(* Logix 5000 project; controller PLC_AutoSeats Emulate 5570 rev 30.12; software revision 30.00 *)

TASK MainTask (continuous, watchdog 500 ms) : MainProgram

MODULES
   Local : Emulate 5570 (ICP 2, rev 30.12)
END_MODULES

VAR_GLOBAL   (* controller tags *)
   Active_PP : BOOL;
   Active_PU : BOOL;
   Active_Soldadura : BOOL;
   Auto : BOOL;
   Emer_Stop_SCADA_PP : BOOL;
   Emer_Stop_SCADA_PU : BOOL;
   Emer_Stop_SCADA_Soldadura : BOOL;
   Estado_PP : DINT;
   Estado_PU : DINT;
   Estado_Soldadura : DINT;
   Mantenimiento_PP : BOOL;
   Mantenimiento_PU : BOOL;
   Mantenimiento_Soldadura : BOOL;
   Manual : BOOL := 1;
   Modo_Op : DINT;
   OSF_01 : BOOL;
   OSF_02 : BOOL;
   OSF_OB_01 : BOOL;
   OSF_OB_02 : BOOL;
   OSR_01 : BOOL;
   OSR_02 : BOOL;
   OSR_03 : BOOL;
   OSR_04 : BOOL;
   OSR_05 : BOOL;
   OSR_06 : BOOL;
   OSR_07 : BOOL;
   OSR_08 : BOOL;
   OSR_09 : BOOL;
   OSR_OB_01 : BOOL;
   OSR_OB_02 : BOOL;
   OSR_OB_03 : BOOL;
   OSR_OB_04 : BOOL;
   OSR_OB_05 : BOOL;
   OSR_OB_06 : BOOL;
   OSR_OB_07 : BOOL;
   OSR_OB_08 : BOOL;
   OSR_OB_09 : BOOL;
   Parar_Ciclo_PP : BOOL;
   Parar_Ciclo_PU : BOOL;
   Parar_Ciclo_Soldadura : BOOL;
   PP_Banda : BOOL;
   PP_Gen_Reposabrazo : BOOL;
   PP_Mover_Molde : BOOL;
   PP_Pos_Molde : REAL;
   PP_Resistencia : BOOL;
   PP_Sensor_Banda_Salida : BOOL;
   PP_Sensor_Molde_Abierto : BOOL;
   PP_Sensor_Molde_Cerrado : BOOL;
   PP_Step1 : BOOL;
   PP_Step2 : BOOL;
   PP_Step3 : BOOL;
   PP_Step4 : BOOL;
   PP_Step5 : BOOL;
   PP_Step6 : BOOL;
   PP_Step7 : BOOL;
   PP_Step8 : BOOL;
   PP_Tornillo_Ext : DINT;
   Producto : DINT;
   PU_Act_Eyector : BOOL;
   PU_Act_Inyector : BOOL;
   PU_Sensor_Pos_MC_1 : DINT;
   PU_Sensor_Pos_MC_2 : DINT;
   PU_Sensor_Pos_ME_1 : DINT;
   PU_Sensor_Pos_ME_2 : DINT;
   PU_Sensor_Pos_R1 : DINT;
   PU_Sensor_Pos_R2 : DINT;
   PU_Sensor_Pos_R3 : DINT;
   Soldadura_Banda_Entrada : BOOL;
   Soldadura_Banda_Salida : BOOL;
   Soldadura_Eli_Marco_Salida : BOOL;
   Soldadura_Eli_Material_Entrada : BOOL;
   Soldadura_Gen_Marco_Salida : BOOL;
   Soldadura_Gen_Material_Entrada : BOOL;
   Soldadura_Giro_0_Listo : BOOL;
   Soldadura_Giro_180_Listo : BOOL;
   Soldadura_Giro_Listo : BOOL;
   Soldadura_Matriz : DINT;
   Soldadura_Primera_Listo : BOOL;
   Soldadura_Segunda_Listo : BOOL;
   Soldadura_Sensor_Entrada : BOOL;
   Soldadura_Sensor_Entrada_Aux : BOOL;
   Soldadura_Sensor_Pos_Matriz : DINT;
   Soldadura_Sensor_Salida : BOOL;
   Soldadura_Sensor_Salida_Aux : BOOL;
   Soldadura_Start_Operario : BOOL;
   Soldadura_Step1 : BOOL;
   Soldadura_Step2 : BOOL;
   Soldadura_Step3 : BOOL;
   Soldadura_Step4 : BOOL;
   Soldadura_Step5 : BOOL;
   Soldadura_Step6 : BOOL;
   Soldadura_Step7 : BOOL;
   Soldadura_Step8 : BOOL;
   Soldadura_Step9 : BOOL;
   Start_Fisico_PP : BOOL;   // Boton Verde Fisico
   Start_Fisico_PU : BOOL;
   Start_Fisico_Soldadura : BOOL;
   Start_SCADA_PP : BOOL;
   Start_SCADA_PU : BOOL;
   Start_SCADA_Soldadura : BOOL;
   Start_Telegram_PP : BOOL;
   Start_Telegram_PU : BOOL;
   Start_Telegram_Soldadura : BOOL;
   Stop_Fisico_PP : BOOL;
   Stop_Fisico_PU : BOOL;
   Stop_Fisico_Soldadura : BOOL;
   Stop_SCADA_PP : BOOL;
   Stop_SCADA_PU : BOOL;
   Stop_SCADA_Soldadura : BOOL;
   Stop_Telegram_PU : BOOL;
   Temp_PP : BOOL;
   Temp_PU : BOOL;
   Temp_Soldadura : BOOL;
   TOF_01 : TIMER := (PRE := 1000);
   TOF_02 : TIMER := (PRE := 1000);
   TOF_03 : TIMER := (PRE := 1000);
   TOF_04 : TIMER := (PRE := 3000);
   TOF_05 : TIMER := (PRE := 1000);
   TOF_06 : TIMER := (PRE := 1000);
   TOF_07 : TIMER := (PRE := 3000);
   TOF_08 : TIMER := (PRE := 1000);
   TON_01 : TIMER := (PRE := 8000);
   TON_02 : TIMER := (PRE := 10000);
   TON_03 : TIMER := (PRE := 10000);
   TON_04 : TIMER := (PRE := 7500);
   TON_05 : TIMER := (PRE := 5000);
END_VAR

PROGRAM MainProgram   (* main routine MainRoutine *)

ROUTINE Celda_Inyeccion_PP   (* ladder *)
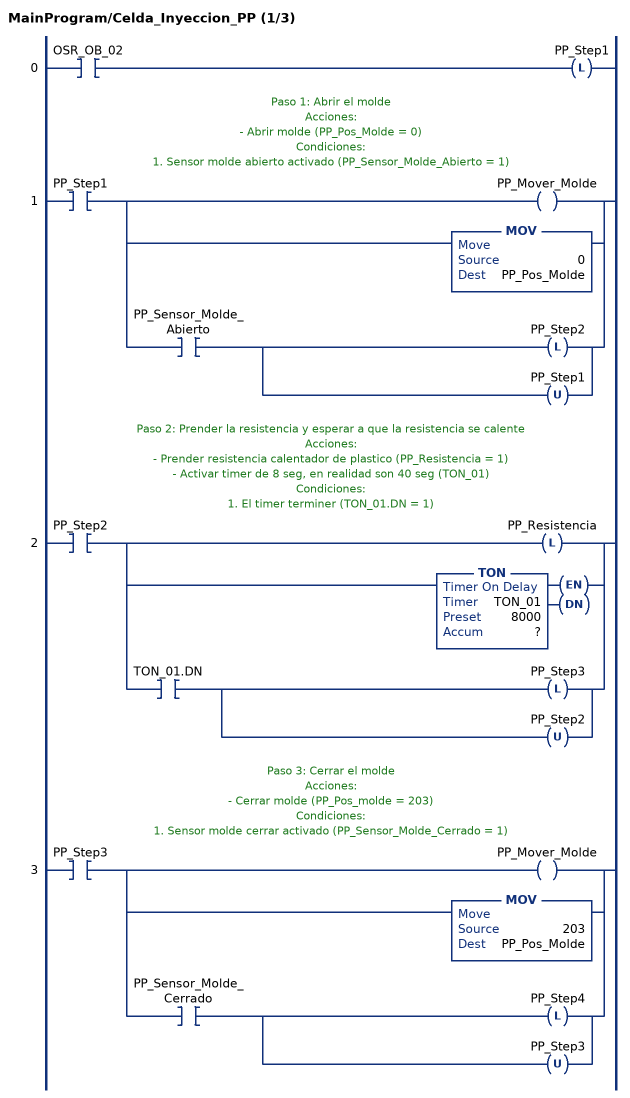
   0: XIC(OSR_OB_02)OTL(PP_Step1);
   // Paso 1: Abrir el molde
   // Acciones:
   // - Abrir molde (PP_Pos_Molde = 0)
   // Condiciones:
   // 1. Sensor molde abierto activado (PP_Sensor_Molde_Abierto = 1)
   1: XIC(PP_Step1)[[OTE(PP_Mover_Molde) ,MOV(0,PP_Pos_Molde) ] ,XIC(PP_Sensor_Molde_Abierto) [OTL(PP_Step2) ,OTU(PP_Step1) ] ];
   // Paso 2: Prender la resistencia y esperar a que la resistencia se calente
   // Acciones:
   // - Prender resistencia calentador de plastico (PP_Resistencia = 1)
   // - Activar timer de 8 seg, en realidad son 40 seg (TON_01)
   // Condiciones:
   // 1. El timer terminer (TON_01.DN = 1)
   2: XIC(PP_Step2)[[OTL(PP_Resistencia) ,TON(TON_01,?,?) ] ,XIC(TON_01.DN) [OTL(PP_Step3) ,OTU(PP_Step2) ] ];
   // Paso 3: Cerrar el molde
   // Acciones:
   // - Cerrar molde (PP_Pos_molde = 203)
   // Condiciones:
   // 1. Sensor molde cerrar activado (PP_Sensor_Molde_Cerrado = 1)
   3: XIC(PP_Step3)[[OTE(PP_Mover_Molde) ,MOV(203,PP_Pos_Molde) ] ,XIC(PP_Sensor_Molde_Cerrado) [OTL(PP_Step4) ,OTU(PP_Step3) ] ];
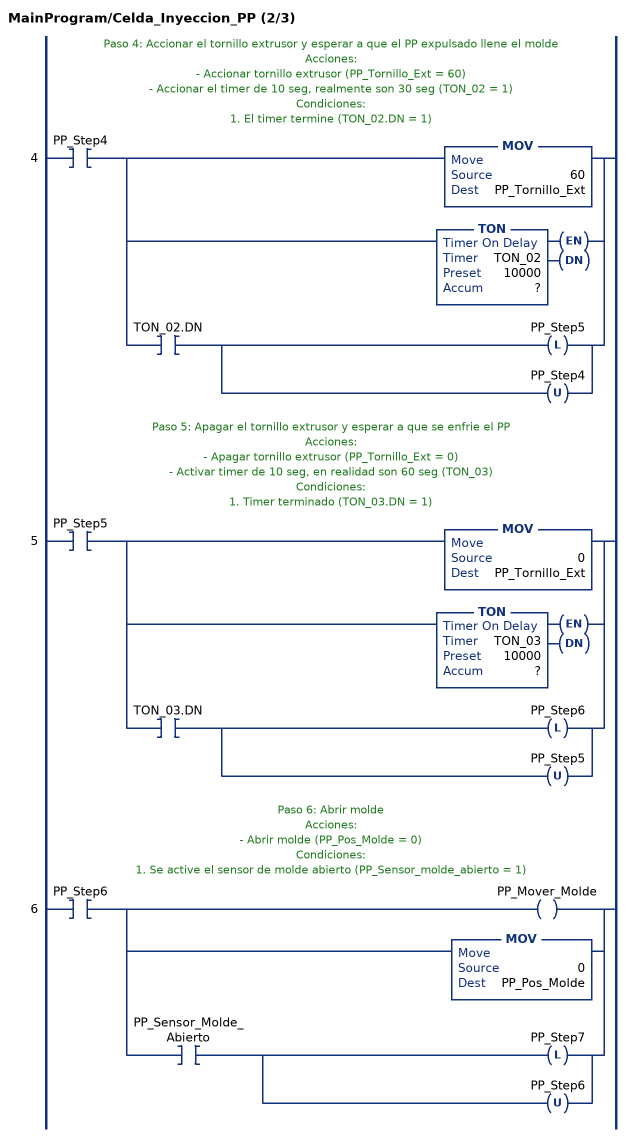
   // Paso 4: Accionar el tornillo extrusor y esperar a que el PP expulsado llene el molde
   // Acciones:
   // - Accionar tornillo extrusor (PP_Tornillo_Ext = 60)
   // - Accionar el timer de 10 seg, realmente son 30 seg (TON_02 = 1)
   // Condiciones:
   // 1. El timer termine (TON_02.DN = 1)
   4: XIC(PP_Step4)[[MOV(60,PP_Tornillo_Ext) ,TON(TON_02,?,?) ] ,XIC(TON_02.DN) [OTL(PP_Step5) ,OTU(PP_Step4) ] ];
   // Paso 5: Apagar el tornillo extrusor y esperar a que se enfrie el PP
   // Acciones:
   // - Apagar tornillo extrusor (PP_Tornillo_Ext = 0)
   // - Activar timer de 10 seg, en realidad son 60 seg (TON_03)
   // Condiciones:
   // 1. Timer terminado (TON_03.DN = 1)
   5: XIC(PP_Step5)[[MOV(0,PP_Tornillo_Ext) ,TON(TON_03,?,?) ] ,XIC(TON_03.DN) [OTL(PP_Step6) ,OTU(PP_Step5) ] ];
   // Paso 6: Abrir molde
   // Acciones:
   // - Abrir molde (PP_Pos_Molde = 0)
   // Condiciones:
   // 1. Se active el sensor de molde abierto (PP_Sensor_molde_abierto = 1)
   6: XIC(PP_Step6)[[OTE(PP_Mover_Molde) ,MOV(0,PP_Pos_Molde) ] ,XIC(PP_Sensor_Molde_Abierto) [OTL(PP_Step7) ,OTU(PP_Step6) ] ];
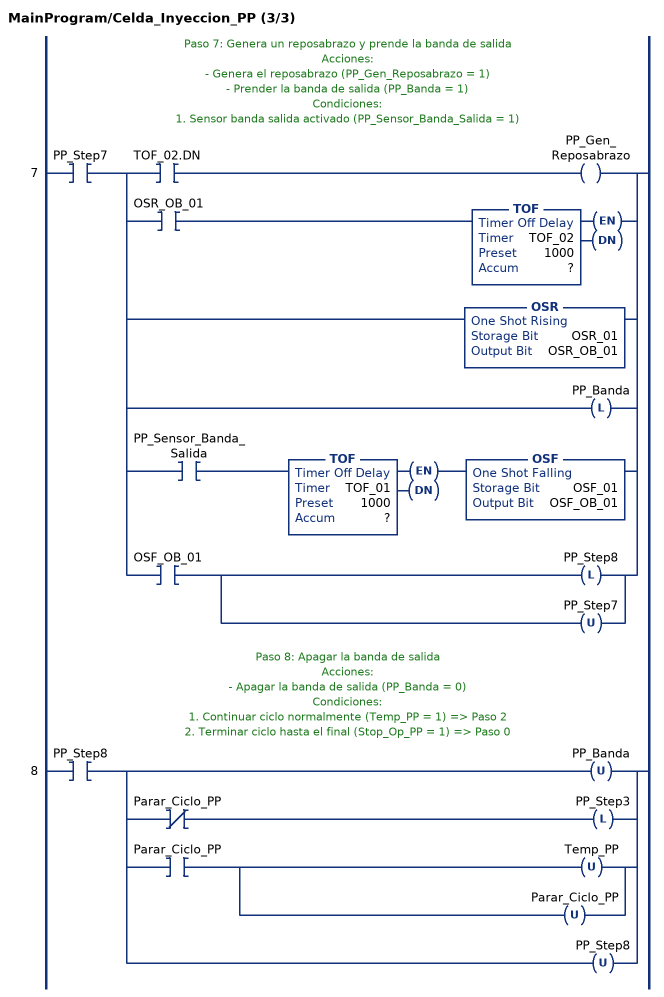
   // Paso 7: Genera un reposabrazo y prende la banda de salida
   // Acciones:
   // - Genera el reposabrazo (PP_Gen_Reposabrazo = 1)
   // - Prender la banda de salida (PP_Banda = 1)
   // Condiciones:
   // 1. Sensor banda salida activado (PP_Sensor_Banda_Salida = 1)
   7: XIC(PP_Step7)[[[[XIC(TOF_02.DN) OTE(PP_Gen_Reposabrazo) ,XIC(OSR_OB_01) TOF(TOF_02,?,?) ] ,OSR(OSR_01,OSR_OB_01) ] ,[OTL(PP_Banda) ,XIC(PP_Sensor_Banda_Salida) TOF(TOF_01,?,?) OSF(OSF_01,OSF_OB_01) ] ] ,XIC(OSF_OB_01) [OTL(PP_Step8) ,OTU(PP_Step7) ] ];
   // Paso 8: Apagar la banda de salida
   // Acciones:
   // - Apagar la banda de salida (PP_Banda = 0)
   // Condiciones:
   // 1. Continuar ciclo normalmente (Temp_PP = 1) => Paso 2
   // 2. Terminar ciclo hasta el final (Stop_Op_PP = 1) => Paso 0
   8: XIC(PP_Step8)[OTU(PP_Banda) ,[[XIO(Parar_Ciclo_PP) OTL(PP_Step3) ,XIC(Parar_Ciclo_PP) [OTU(Temp_PP) ,OTU(Parar_Ciclo_PP) ] ] ,OTU(PP_Step8) ] ];
END_ROUTINE

ROUTINE Celda_Soldadura   (* ladder *)
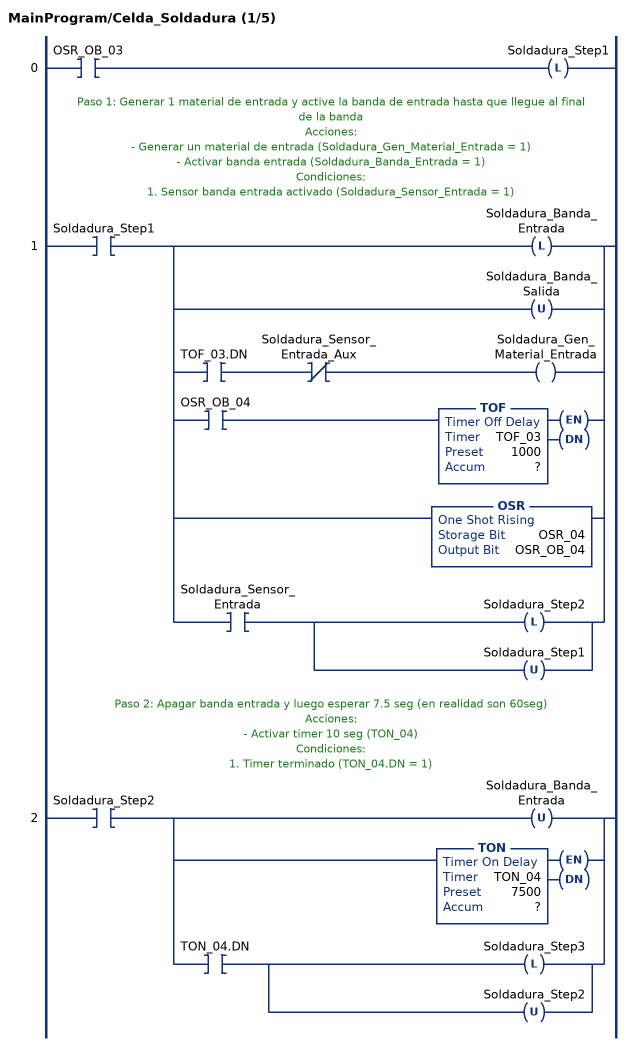
   0: XIC(OSR_OB_03)OTL(Soldadura_Step1);
   // Paso 1: Generar 1 material de entrada y active la banda de entrada hasta que llegue al final de la banda
   // Acciones:
   // - Generar un material de entrada (Soldadura_Gen_Material_Entrada = 1)
   // - Activar banda entrada (Soldadura_Banda_Entrada = 1)
   // Condiciones:
   // 1. Sensor banda entrada activado (Soldadura_Sensor_Entrada = 1)
   1: XIC(Soldadura_Step1)[[[OTL(Soldadura_Banda_Entrada) ,OTU(Soldadura_Banda_Salida) ] ,[XIC(TOF_03.DN) XIO(Soldadura_Sensor_Entrada_Aux) OTE(Soldadura_Gen_Material_Entrada) ,[XIC(OSR_OB_04) TOF(TOF_03,?,?) ,OSR(OSR_04,OSR_OB_04) ] ] ] ,XIC(Soldadura_Sensor_Entrada) [OTL(Soldadura_Step2) ,OTU(Soldadura_Step1) ] ];
   // Paso 2: Apagar banda entrada y luego esperar 7.5 seg (en realidad son 60seg)
   // Acciones:
   // - Activar timer 10 seg (TON_04)
   // Condiciones:
   // 1. Timer terminado (TON_04.DN = 1)
   2: XIC(Soldadura_Step2)[[OTU(Soldadura_Banda_Entrada) ,TON(TON_04,?,?) ] ,XIC(TON_04.DN) [OTL(Soldadura_Step3) ,OTU(Soldadura_Step2) ] ];
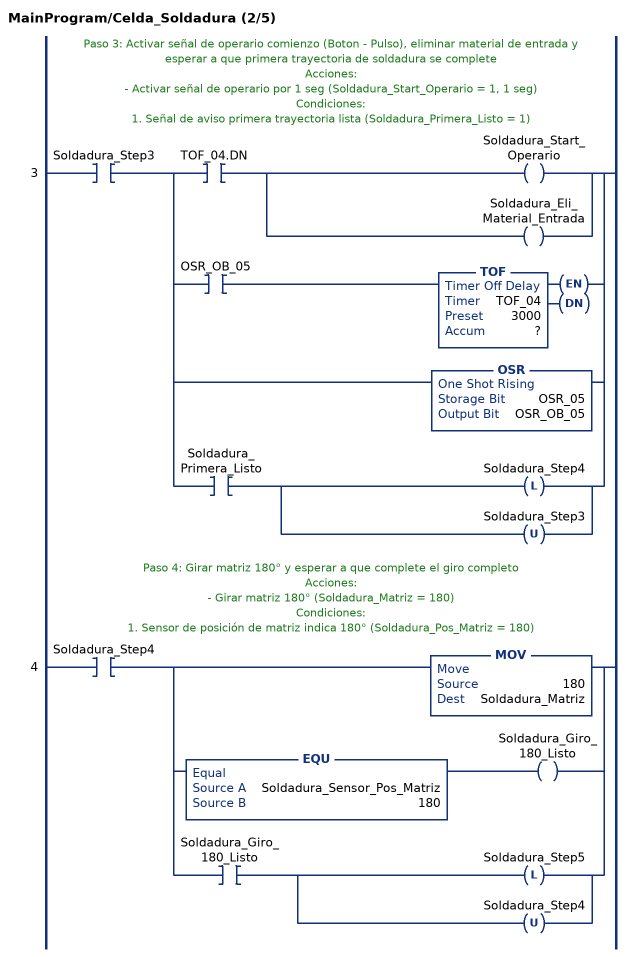
   // Paso 3: Activar señal de operario comienzo (Boton - Pulso), eliminar material de entrada y esperar a que primera trayectoria de soldadura se complete
   // Acciones:
   // - Activar señal de operario por 1 seg (Soldadura_Start_Operario = 1, 1 seg)
   // Condiciones:
   // 1. Señal de aviso primera trayectoria lista (Soldadura_Primera_Listo = 1)
   3: XIC(Soldadura_Step3)[[XIC(TOF_04.DN) [OTE(Soldadura_Start_Operario) ,OTE(Soldadura_Eli_Material_Entrada) ] ,[XIC(OSR_OB_05) TOF(TOF_04,?,?) ,OSR(OSR_05,OSR_OB_05) ] ] ,XIC(Soldadura_Primera_Listo) [OTL(Soldadura_Step4) ,OTU(Soldadura_Step3) ] ];
   // Paso 4: Girar matriz 180° y esperar a que complete el giro completo
   // Acciones:
   // - Girar matriz 180° (Soldadura_Matriz = 180)
   // Condiciones:
   // 1. Sensor de posición de matriz indica 180° (Soldadura_Pos_Matriz = 180)
   4: XIC(Soldadura_Step4)[[MOV(180,Soldadura_Matriz) ,EQU(Soldadura_Sensor_Pos_Matriz,180) OTE(Soldadura_Giro_180_Listo) ] ,XIC(Soldadura_Giro_180_Listo) [OTL(Soldadura_Step5) ,OTU(Soldadura_Step4) ] ];
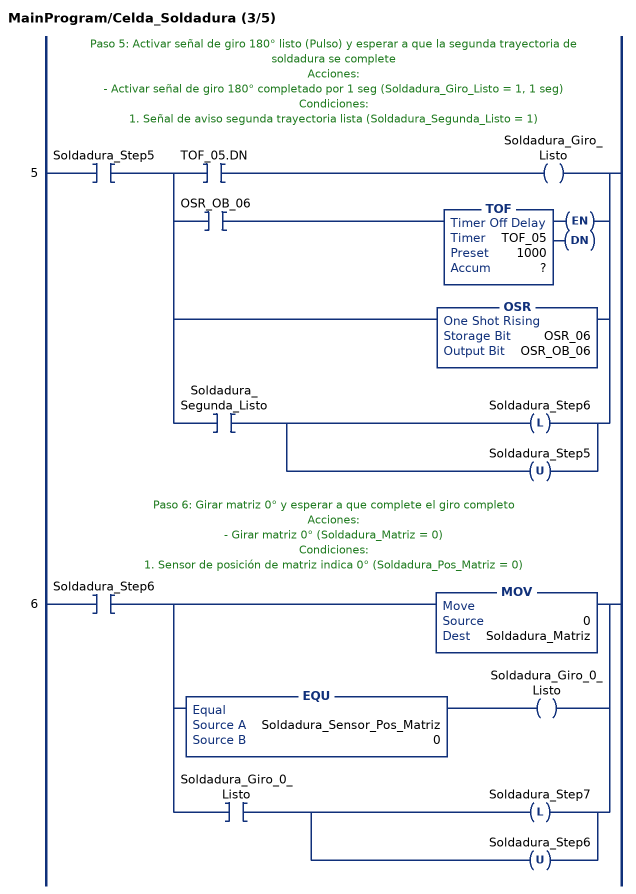
   // Paso 5: Activar señal de giro 180° listo (Pulso) y esperar a que la segunda trayectoria de soldadura se complete
   // Acciones:
   // - Activar señal de giro 180° completado por 1 seg (Soldadura_Giro_Listo = 1, 1 seg)
   // Condiciones:
   // 1. Señal de aviso segunda trayectoria lista (Soldadura_Segunda_Listo = 1)
   5: XIC(Soldadura_Step5)[[XIC(TOF_05.DN) OTE(Soldadura_Giro_Listo) ,[XIC(OSR_OB_06) TOF(TOF_05,?,?) ,OSR(OSR_06,OSR_OB_06) ] ] ,XIC(Soldadura_Segunda_Listo) [OTL(Soldadura_Step6) ,OTU(Soldadura_Step5) ] ];
   // Paso 6: Girar matriz 0° y esperar a que complete el giro completo
   // Acciones:
   // - Girar matriz 0° (Soldadura_Matriz = 0)
   // Condiciones:
   // 1. Sensor de posición de matriz indica 0° (Soldadura_Pos_Matriz = 0)
   6: XIC(Soldadura_Step6)[[MOV(0,Soldadura_Matriz) ,EQU(Soldadura_Sensor_Pos_Matriz,0) OTE(Soldadura_Giro_0_Listo) ] ,XIC(Soldadura_Giro_0_Listo) [OTL(Soldadura_Step7) ,OTU(Soldadura_Step6) ] ];
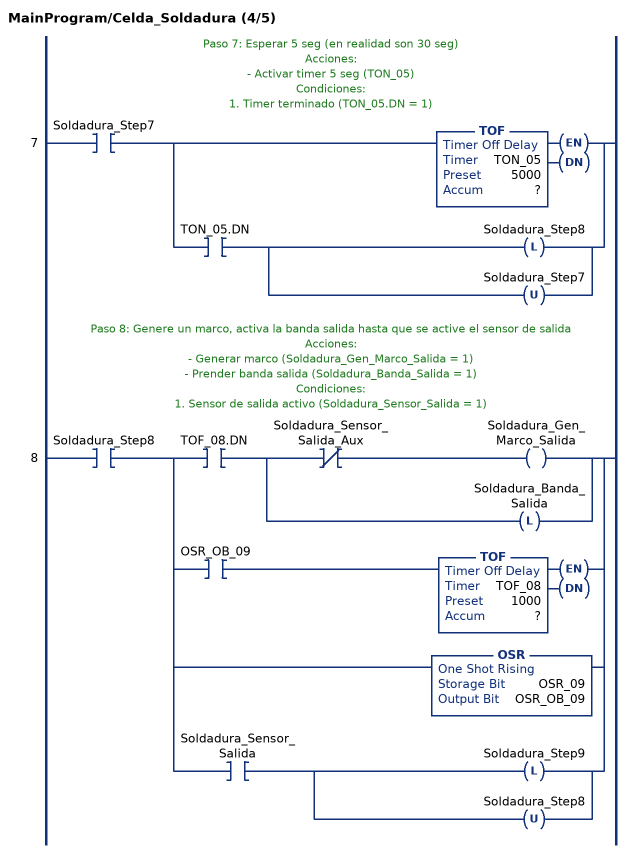
   // Paso 7: Esperar 5 seg (en realidad son 30 seg)
   // Acciones:
   // - Activar timer 5 seg (TON_05)
   // Condiciones:
   // 1. Timer terminado (TON_05.DN = 1)
   7: XIC(Soldadura_Step7)[TOF(TON_05,?,?) ,XIC(TON_05.DN) [OTL(Soldadura_Step8) ,OTU(Soldadura_Step7) ] ];
   // Paso 8: Genere un marco, activa la banda salida hasta que se active el sensor de salida
   // Acciones:
   // - Generar marco (Soldadura_Gen_Marco_Salida = 1)
   // - Prender banda salida (Soldadura_Banda_Salida = 1)
   // Condiciones:
   // 1. Sensor de salida activo (Soldadura_Sensor_Salida = 1)
   8: XIC(Soldadura_Step8)[[XIC(TOF_08.DN) [XIO(Soldadura_Sensor_Salida_Aux) OTE(Soldadura_Gen_Marco_Salida) ,OTL(Soldadura_Banda_Salida) ] ,[XIC(OSR_OB_09) TOF(TOF_08,?,?) ,OSR(OSR_09,OSR_OB_09) ] ] ,XIC(Soldadura_Sensor_Salida) [OTL(Soldadura_Step9) ,OTU(Soldadura_Step8) ] ];
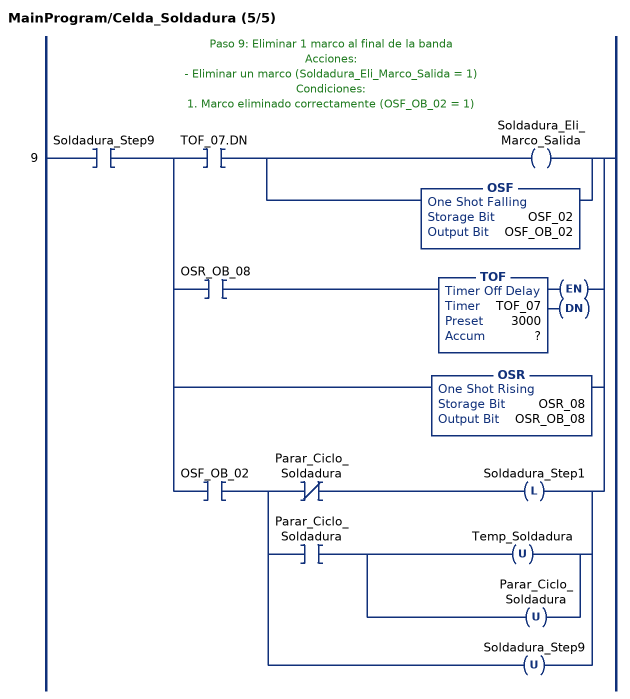
   // Paso 9: Eliminar 1 marco al final de la banda
   // Acciones:
   // - Eliminar un marco (Soldadura_Eli_Marco_Salida = 1)
   // Condiciones:
   // 1. Marco eliminado correctamente (OSF_OB_02 = 1)
   9: XIC(Soldadura_Step9)[[XIC(TOF_07.DN) [OTE(Soldadura_Eli_Marco_Salida) ,OSF(OSF_02,OSF_OB_02) ] ,[XIC(OSR_OB_08) TOF(TOF_07,?,?) ,OSR(OSR_08,OSR_OB_08) ] ] ,XIC(OSF_OB_02) [[XIO(Parar_Ciclo_Soldadura) OTL(Soldadura_Step1) ,XIC(Parar_Ciclo_Soldadura) [OTU(Temp_Soldadura) ,OTU(Parar_Ciclo_Soldadura) ] ] ,OTU(Soldadura_Step9) ] ];
END_ROUTINE

ROUTINE Control_Celda_Inyeccion_PP   (* ladder *)
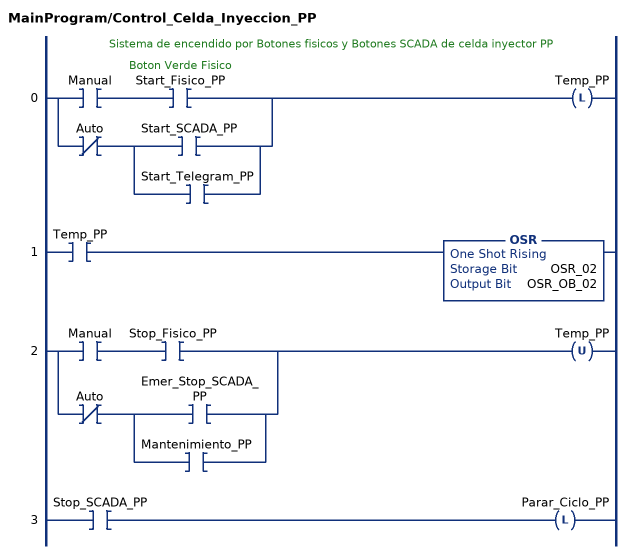
   // Sistema de encendido por Botones fisicos y Botones SCADA de celda inyector PP
   0: [XIC(Manual) XIC(Start_Fisico_PP) ,XIO(Auto) [XIC(Start_SCADA_PP) ,XIC(Start_Telegram_PP) ] ]OTL(Temp_PP);
   1: XIC(Temp_PP)OSR(OSR_02,OSR_OB_02);
   2: [XIC(Manual) XIC(Stop_Fisico_PP) ,XIO(Auto) [XIC(Emer_Stop_SCADA_PP) ,XIC(Mantenimiento_PP) ] ]OTU(Temp_PP);
   3: XIC(Stop_SCADA_PP)OTL(Parar_Ciclo_PP);
END_ROUTINE

ROUTINE Control_Celda_Moldeo_PU   (* ladder *)
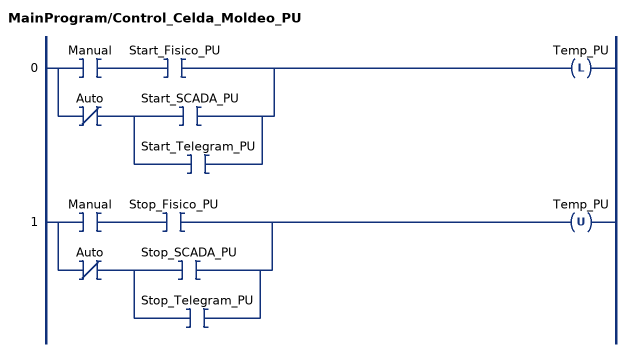
   0: [XIC(Manual) XIC(Start_Fisico_PU) ,XIO(Auto) [XIC(Start_SCADA_PU) ,XIC(Start_Telegram_PU) ] ]OTL(Temp_PU);
   1: [XIC(Manual) XIC(Stop_Fisico_PU) ,XIO(Auto) [XIC(Stop_SCADA_PU) ,XIC(Stop_Telegram_PU) ] ]OTU(Temp_PU);
END_ROUTINE

ROUTINE Control_Celda_Soldadura   (* ladder *)
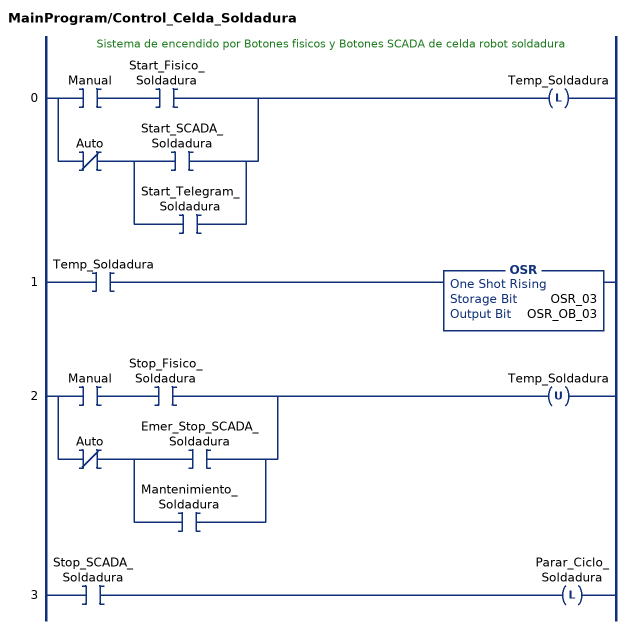
   // Sistema de encendido por Botones fisicos y Botones SCADA de celda robot soldadura
   0: [XIC(Manual) XIC(Start_Fisico_Soldadura) ,XIO(Auto) [XIC(Start_SCADA_Soldadura) ,XIC(Start_Telegram_Soldadura) ] ]OTL(Temp_Soldadura);
   1: XIC(Temp_Soldadura)OSR(OSR_03,OSR_OB_03);
   2: [XIC(Manual) XIC(Stop_Fisico_Soldadura) ,XIO(Auto) [XIC(Emer_Stop_SCADA_Soldadura) ,XIC(Mantenimiento_Soldadura) ] ]OTU(Temp_Soldadura);
   3: XIC(Stop_SCADA_Soldadura)OTL(Parar_Ciclo_Soldadura);
END_ROUTINE

ROUTINE MainRoutine   (* ladder *)
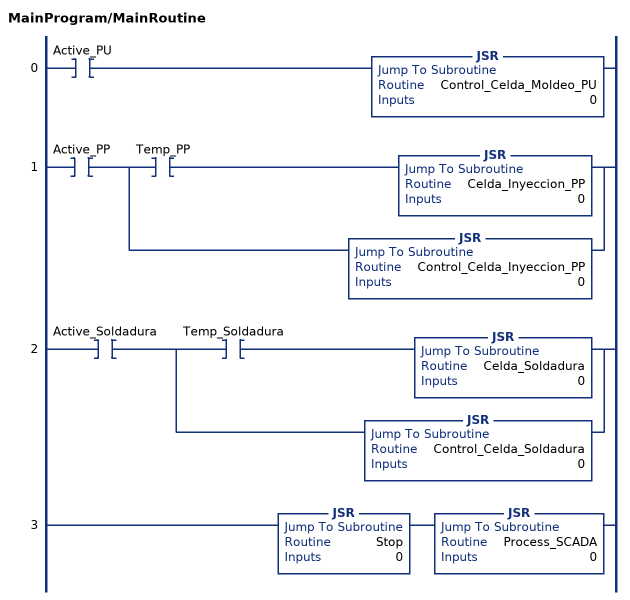
   0: XIC(Active_PU)JSR(Control_Celda_Moldeo_PU,0);
   1: XIC(Active_PP)[XIC(Temp_PP) JSR(Celda_Inyeccion_PP,0) ,JSR(Control_Celda_Inyeccion_PP,0) ];
   2: XIC(Active_Soldadura)[XIC(Temp_Soldadura) JSR(Celda_Soldadura,0) ,JSR(Control_Celda_Soldadura,0) ];
   3: JSR(Stop,0)JSR(Process_SCADA,0);
END_ROUTINE

ROUTINE Process_SCADA   (* ladder *)
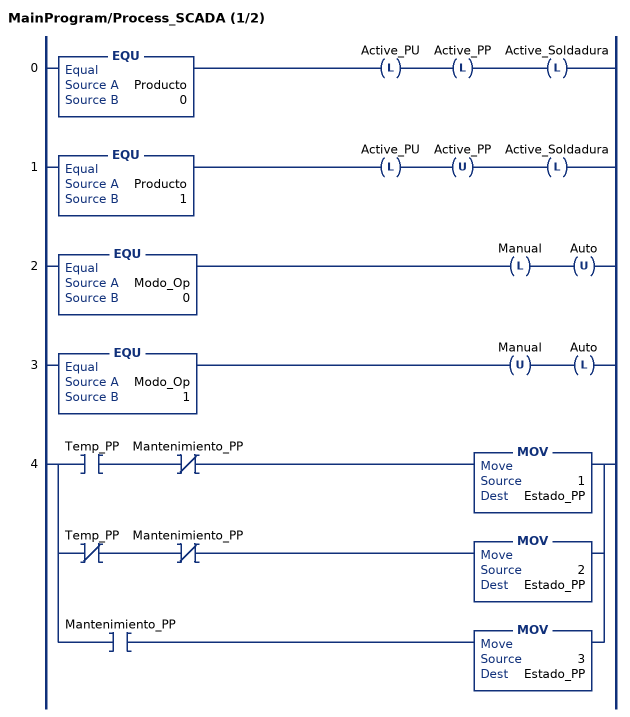
   0: EQU(Producto,0)OTL(Active_PU)OTL(Active_PP)OTL(Active_Soldadura);
   1: EQU(Producto,1)OTL(Active_PU)OTU(Active_PP)OTL(Active_Soldadura);
   2: EQU(Modo_Op,0)OTL(Manual)OTU(Auto);
   3: EQU(Modo_Op,1)OTU(Manual)OTL(Auto);
   4: [XIC(Temp_PP) XIO(Mantenimiento_PP) MOV(1,Estado_PP) ,[XIO(Temp_PP) XIO(Mantenimiento_PP) MOV(2,Estado_PP) ,XIC(Mantenimiento_PP) MOV(3,Estado_PP) ] ];
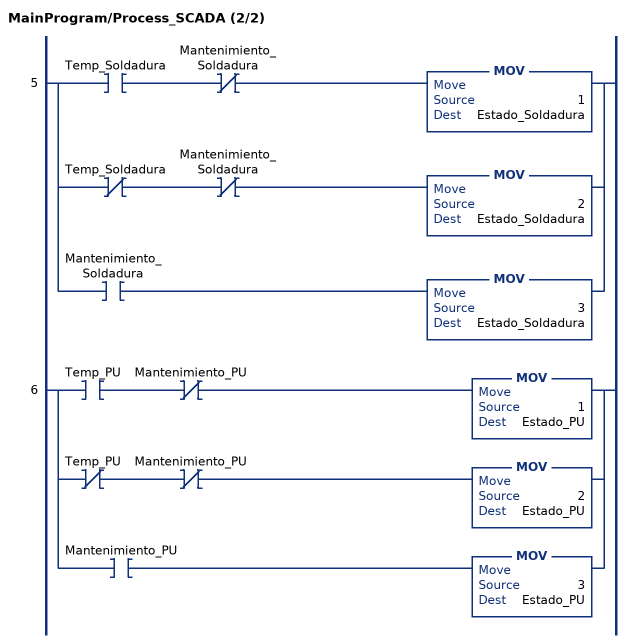
   5: [XIC(Temp_Soldadura) XIO(Mantenimiento_Soldadura) MOV(1,Estado_Soldadura) ,[XIO(Temp_Soldadura) XIO(Mantenimiento_Soldadura) MOV(2,Estado_Soldadura) ,XIC(Mantenimiento_Soldadura) MOV(3,Estado_Soldadura) ] ];
   6: [XIC(Temp_PU) XIO(Mantenimiento_PU) MOV(1,Estado_PU) ,[XIO(Temp_PU) XIO(Mantenimiento_PU) MOV(2,Estado_PU) ,XIC(Mantenimiento_PU) MOV(3,Estado_PU) ] ];
END_ROUTINE

ROUTINE Stop   (* structured text *)
   IF (not Temp_PP) THEN
   	PP_Step1 := 0;
   	PP_Step2 := 0;
   	PP_Step3 := 0;
   	PP_Step4 := 0;
   	PP_Step5 := 0;
   	PP_Step6 := 0;
   	PP_Step7 := 0;
   	PP_Step8 := 0;
   	PP_Resistencia :=0;
   	PP_Banda := 0;
   	PP_Gen_Reposabrazo := 0;
   	PP_Tornillo_Ext := 0;
   END_IF;
   
   IF (not Temp_Soldadura) THEN
   	Soldadura_Step1 := 0;
   	Soldadura_Step2 := 0;
   	Soldadura_Step3 := 0;
   	Soldadura_Step4 := 0;
   	Soldadura_Step5 := 0;
   	Soldadura_Step6 := 0;
   	Soldadura_Step7 := 0;
   	Soldadura_Step8 := 0;
   	Soldadura_Step9 := 0;
   	Soldadura_Banda_Entrada := 0;
   	Soldadura_Banda_Salida := 0;
   	Soldadura_Matriz := Soldadura_Sensor_Pos_Matriz;
   	Soldadura_Gen_Marco_Salida := 0;
   	Soldadura_Gen_Material_Entrada := 0;
   	Soldadura_Eli_Marco_Salida := 0;
   	Soldadura_Eli_Material_Entrada := 0;
   	Soldadura_Start_Operario := 0;
   	Soldadura_Giro_Listo := 0;
   END_IF;
END_ROUTINE
END_PROGRAM
